SUBAPPLICATION Uebung_032 (* LED Strip Blinkende LED *)
  (* Standard: 61499-2 *)
  (* Version 1.0, 2023-10-23, franz *)
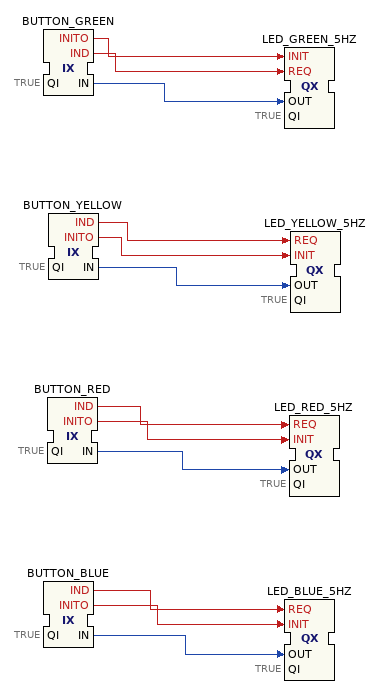
  FBS
    LED_GREEN_5HZ : QX(QI := TRUE);
    BUTTON_GREEN : IX(QI := TRUE);
    BUTTON_YELLOW : IX(QI := TRUE);
    LED_YELLOW_5HZ : QX(QI := TRUE);
    BUTTON_RED : IX(QI := TRUE);
    LED_RED_5HZ : QX(QI := TRUE);
    BUTTON_BLUE : IX(QI := TRUE);
    LED_BLUE_5HZ : QX(QI := TRUE);
  END_FBS
  EVENT_CONNECTIONS
    BUTTON_GREEN.INITO TO LED_GREEN_5HZ.INIT;
    BUTTON_GREEN.IND TO LED_GREEN_5HZ.REQ;
    BUTTON_YELLOW.IND TO LED_YELLOW_5HZ.REQ;
    BUTTON_YELLOW.INITO TO LED_YELLOW_5HZ.INIT;
    BUTTON_RED.IND TO LED_RED_5HZ.REQ;
    BUTTON_RED.INITO TO LED_RED_5HZ.INIT;
    BUTTON_BLUE.IND TO LED_BLUE_5HZ.REQ;
    BUTTON_BLUE.INITO TO LED_BLUE_5HZ.INIT;
  END_CONNECTIONS
  DATA_CONNECTIONS
    BUTTON_GREEN.IN TO LED_GREEN_5HZ.OUT;
    BUTTON_YELLOW.IN TO LED_YELLOW_5HZ.OUT;
    BUTTON_RED.IN TO LED_RED_5HZ.OUT;
    BUTTON_BLUE.IN TO LED_BLUE_5HZ.OUT;
  END_CONNECTIONS
END_SUBAPPLICATION
